TYPE DUT_MotorDriverCommand : STRUCT
    ControlWord  : WORD;
    TargetTorque : INT;
END_STRUCT
END_TYPE

(* stored: Version 1.1.0.1, ProductVersion 3.1.4024.12
   DUT DUT_MotorDriverCommand: Id {9f95b821-e6f9-4e51-98dd-900047a03010} *)
